// TIA Portal project "bientan" (V14)

(* hardware
DEVICE "S7-1200 station_1"  S7-1200 Station
   slot 0: "Rack_0"  S7-1200 Rack  Rack  V1.0
   slot 1: "PLC_1"  CPU 1212C DC/DC/DC  6ES7 212-1AE40-0XB0  V4.2
   slot 3: "CB 1241 (RS485)"  CB 1241 (RS485)  6ES7 241-1CH30-1XB0  V1.0
DEVICE "HMI_1"  KTP400 Basic PN
   slot 0: "KTP400 Basic PN"  KTP400 Basic PN  6AV2 123-2DB03-0AX0  14.0.1.0
   slot 1: "HMI_RT_1"  KTP400 Basic PN  6AV2 123-2DB03-0AX0  14.0.1.0
   slot 5: "HMI_1.IE_CP_1"  PROFINET Interface  14.0.1.0
      slot 1: "PROFINET Interface_1"  PROFINET Interface
         slot 1: "Port_1"  Port
*)

// ===== PLC "PLC_1"  CPU 1212C DC/DC/DC =====

VAR_GLOBAL   // PLC tag table "Default tag table"
   "System_Byte" AT %MB1 : Byte;
   "FirstScan" AT %M1.0 : Bool;
   "DiagStatusUpdate" AT %M1.1 : Bool;
   "AlwaysTRUE" AT %M1.2 : Bool;
   "AlwaysFALSE" AT %M1.3 : Bool;
   "ready" AT %M0.0 : Bool;
   "Tag_2" AT %MW50 : Int;
   "stop" AT %M0.1 : Bool;
   "start" AT %M0.2 : Bool;
   "on" AT %M0.3 : Bool;
   "tan so" AT %M0.4 : Bool;
   "Tag_3" AT %MW1 : Int;
   "tan so 2" AT %M0.5 : Bool;
   "nhap hmi" AT %MD4 : DInt;
END_VAR

ORGANIZATION_BLOCK "Main"   // OB1, LAD, ProgramCycle
TITLE = "Main Program Sweep (Cycle)"
{ S7_Optimized_Access := 'TRUE' }
VERSION : 0.1
   VAR_INPUT
      Initial_Call : Bool;   // Initial call of this OB
      Remanence : Bool;   // =True, if remanent data are available
   END_VAR
BEGIN

REGION Network 1: khoi tao truyen thong
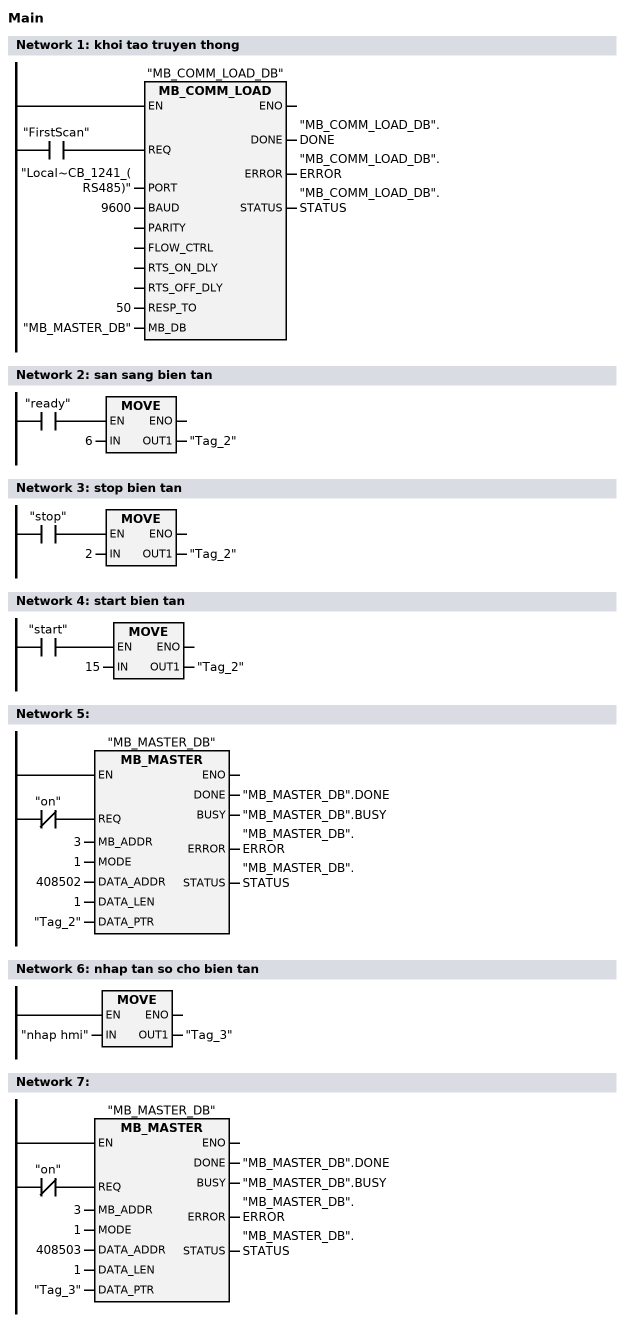
   "MB_COMM_LOAD_DB"(REQ := "FirstScan",   // MB_COMM_LOAD
                     PORT := "Local~CB_1241_(RS485)",
                     BAUD := 9600,
                     RESP_TO := 50,
                     MB_DB := "MB_MASTER_DB",
                     DONE => "MB_COMM_LOAD_DB".DONE,
                     ERROR => "MB_COMM_LOAD_DB".ERROR,
                     STATUS => "MB_COMM_LOAD_DB".STATUS);
END_REGION

REGION Network 2: san sang bien tan
   RUNG wire#powerrail
      Contact( "ready" )
      Move(in := 6, out1 => "Tag_2")
   END_RUNG
   // the same network as SCL:
   IF "ready" THEN "Tag_2" := 6; END_IF;
END_REGION

REGION Network 3: stop bien tan
   RUNG wire#powerrail
      Contact( "stop" )
      Move(in := 2, out1 => "Tag_2")
   END_RUNG
   // the same network as SCL:
   IF "stop" THEN "Tag_2" := 2; END_IF;
END_REGION

REGION Network 4: start bien tan
   RUNG wire#powerrail
      Contact( "start" )
      Move(in := 15, out1 => "Tag_2")
   END_RUNG
   // the same network as SCL:
   IF "start" THEN "Tag_2" := 15; END_IF;
END_REGION

REGION Network 5
   "MB_MASTER_DB"(REQ := NOT "on",   // MB_MASTER
                  MB_ADDR := 3,
                  MODE := 1,
                  DATA_ADDR := 408502,
                  DATA_LEN := 1,
                  DATA_PTR := "Tag_2",
                  DONE => "MB_MASTER_DB".DONE,
                  BUSY => "MB_MASTER_DB".BUSY,
                  ERROR => "MB_MASTER_DB".ERROR,
                  STATUS => "MB_MASTER_DB".STATUS);
END_REGION

REGION Network 6: nhap tan so cho bien tan
   RUNG wire#powerrail
      Move(in := "nhap hmi", out1 => "Tag_3")
   END_RUNG
   // the same network as SCL:
   "Tag_3" := "nhap hmi";
END_REGION

REGION Network 7
   "MB_MASTER_DB"(REQ := NOT "on",   // MB_MASTER
                  MB_ADDR := 3,
                  MODE := 1,
                  DATA_ADDR := 408503,
                  DATA_LEN := 1,
                  DATA_PTR := "Tag_3",
                  DONE => "MB_MASTER_DB".DONE,
                  BUSY => "MB_MASTER_DB".BUSY,
                  ERROR => "MB_MASTER_DB".ERROR,
                  STATUS => "MB_MASTER_DB".STATUS);
END_REGION
END_ORGANIZATION_BLOCK

(* ===== HMI "HMI_RT_1" =====
system functions are stored by id; their names below are inferred from use
connection "HMI_Connection_1": ETHERNET, SMART_S7_1200_OMS

HMI tags "Default tag table"
   "start" : Bool = PLC start AT %M0.2, 100 ms
   "stop" : Bool = PLC stop AT %M0.1, 100 ms
   "ready" : Bool = PLC ready AT %M0.0, 100 ms
   "nhap hmi" : DInt = PLC "nhap hmi" AT %MD4, 100 ms

Template "Template_1" 480x272
   Button "Exit" at 388,227 size 63x44; TextOff 'Exit'; PictureOff "ExitRuntime_KTP400_Basic_PN_TR"; PictureOn "ExitRuntime_KTP400_Basic_PN_TR"
      on Release: StopRuntime(0)
   Button "Template_Button" at 268,227 size 63x44; TextOff 'Text'
   Button "Template_Button_1" at 148,227 size 63x44; TextOff 'Text'
   Button "Start screen" at 28,227 size 63x44; TextOff 'Start screen'; PictureOff "NavigateHome_KTP400_Basic_PN_TR"; PictureOn "NavigateHome_KTP400_Basic_PN_TR"
      on Release: ActivateScreen("Root screen", 0)

screen "Root screen" 480x272, template "Template_1"
   TextField "HmiScreenItemData" at 46,19 size 384x22; Text 'TRUYEN THONG PLC BIEN TAN VA HMI'
   Button "Button_1" at 42,143 size 96x32; TextOff 'READY'
      on Press: SetBit("ready")
      on Release: ResetBit("ready")
   Button "Button_2" at 204,140 size 96x32; TextOff 'START'
      on Press: SetBit("start")
      on Release: ResetBit("start")
   Button "Button_3" at 369,139 size 96x32; TextOff 'STOP'
      on Press: SetBit("stop")
      on Release: ResetBit("stop")
   IOField "I/O field_1" at 203,73 size 96x32; FormatPattern s9999999999
      ProcessValue <- "nhap hmi"
*)